// TwinCAT 3 PLC project FluentCode
// ProgramVersion: 3.1.4023.0
// libraries:
//   Tc2_Standard, * (Beckhoff Automation GmbH)
//   Tc2_System, * (Beckhoff Automation GmbH)
//   Tc2_Utilities, * (Beckhoff Automation GmbH)
//   Tc3_Module, * (Beckhoff Automation GmbH)
// project tree:
//   / PlcTask.TcTTO
//   POUs/ ILimitedStringBuilder.TcIO, IStringBuilder.TcIO, MAIN.TcPOU, StringBuilder.TcPOU
// real-time tasks:
//   TASK PlcTask: cycle T#10ms, priority 20, ADS port 350

CONFIGURATION FluentCode
    RESOURCE PLC ON TwinCAT3
        TASK PlcTask(INTERVAL := T#10ms, PRIORITY := 20);
        PROGRAM MAIN WITH PlcTask : MAIN;
    END_RESOURCE
END_CONFIGURATION

// ---- POUs/ILimitedStringBuilder.TcIO
INTERFACE ILimitedStringBuilder

METHOD  Append : IStringBuilder // Append text to t current build string.
VAR_INPUT
	text:STRING; //Text to append to current build string
END_VAR
END_METHOD

METHOD Reset : ILimitedStringBuilder //Reset current build string to an empty string.
END_METHOD

METHOD ToString : STRING //Returns current build string.
END_METHOD

END_INTERFACE

// ---- POUs/IStringBuilder.TcIO
INTERFACE IStringBuilder

METHOD  Append : IStringBuilder // Append text to t current build string.
VAR_INPUT
	text:STRING; //Text to append to current build string
END_VAR
END_METHOD

METHOD InsertAtLocation : IStringBuilder
VAR_INPUT
	Text:STRING;
	Position:INT;
END_VAR
END_METHOD

METHOD Reset : ILimitedStringBuilder //Reset current build string to an empty string.
END_METHOD

METHOD ToString : STRING //Returns current build string.
END_METHOD

END_INTERFACE

// ---- POUs/MAIN.TcPOU
PROGRAM MAIN
VAR
	ErrorString_WithConcat:STRING;
	ErrorString_WithFluentCode:STRING;
	ErrorMessage:STRING := 'Important message';
	ErrorNumber:int := 1;
	_StringBuilder:StringBuilder;
	StringAreEqual:BOOL;
	StringAreStillEqual:BOOL;
END_VAR

ErrorString_WithConcat := CONCAT(CONCAT(CONCAT(CONCAT('Error number: ' , INT_TO_STRING(ErrorNumber)),'. Message: '),ErrorMessage),'.');
ErrorString_WithConcat := Concat('Error number: ' , INT_TO_STRING(ErrorNumber));
ErrorString_WithConcat := Concat(ErrorString_WithConcat , '. Message: ');
ErrorString_WithConcat := Concat(ErrorString_WithConcat , ErrorMessage);
ErrorString_WithConcat := Concat(ErrorString_WithConcat , '.');
							
ErrorString_WithFluentCode := _StringBuilder.Reset()
							.Append('Error number: ')
							.Append(INT_TO_STRING(ErrorNumber))
							.Append('. Message: ')
							.Append(ErrorMessage)
							.Append('.')
							.ToString();
							
StringAreEqual := ErrorString_WithConcat = ErrorString_WithFluentCode;

ErrorString_WithConcat := INSERT( ErrorString_WithConcat, ' extended',43);
ErrorString_WithFluentCode := _StringBuilder.InsertAtLocation(' extended',43).ToString();

StringAreStillEqual :=  ErrorString_WithConcat = ErrorString_WithFluentCode;

END_PROGRAM

// ---- POUs/StringBuilder.TcPOU
FUNCTION_BLOCK PUBLIC StringBuilder IMPLEMENTS  IStringBuilder, ILimitedStringBuilder
VAR
	{attribute 'hide'}
	_workString:STRING;
END_VAR

METHOD PUBLIC Append : IStringBuilder // Append text to t current build string.
VAR_INPUT
	text:STRING; //Text to append to current build string
END_VAR
_workString:= Concat(_workString,text);
Append := THIS^;
END_METHOD

METHOD PUBLIC InsertAtLocation : IStringBuilder
VAR_INPUT
	Text:STRING;
	Position:INT;
END_VAR
_workString := Tc2_Standard.INSERT(_WorkSTring,Text,Position);
InsertAtLocation  := THIS^;
END_METHOD

METHOD PUBLIC Reset : ILimitedStringBuilder //Reset current build string to an empty string.
_workString:='';
Reset := THIS^;
END_METHOD

METHOD PUBLIC ToString : STRING //Returns current build string.
ToString := _workString;
END_METHOD

END_FUNCTION_BLOCK
